(* Logix 5000 project; controller MetsoFilter vendor 1 type 14 code 106 rev 32.11; software revision 32.00 *)

TASK MainTask (continuous, watchdog 500 ms) : MainProgram

MODULES
   Local : vendor 1 type 14 code 106 (Compact 0, rev 32.11)
END_MODULES

TYPE Status_Cycle :   // Status for Each Cycle
STRUCT
   Start_Time : STRING;   // Start Time of Cycle HH:MM
   Cycle_Time : INT;   // Cycle Time in Seconds
   Press_Weight : INT;   // Press wieght of Cycle in Kg
   Pump_Time : INT;   // Pump time in Seconds
   Drying_Time : INT;   // Drying time in Seconds
END_STRUCT
END_TYPE

TYPE Status_Day :   // Status for Each Day
STRUCT
   Date : STRING;   // Days Date
   Total_Tons : REAL;   // Total Tons for the Day
   Shift1_Tons : REAL;   // Shift #1 tons
   Shift2_Tons : REAL;   // Shift #2 Tons
   Shift3_Tons : REAL;   // Shift #3 tons
END_STRUCT
END_TYPE

VAR_GLOBAL   (* controller tags *)
   Alarm_Hatches : BOOL;   // Hatches have taken too long to open or close
   AlarmHornPulser : BOOL;   // Pulse Horn during a new alarm
   AlarmReset : BOOL;   // Alarm Rest Relay
   ALM_AirAndWaterOK_T : TIMER;   // Air and Water OK, Enable Air & Water Valves Alarms
   ALM_DryAir : BOOL;   // Dry Air Not OK
   ALM_LowBattery : BOOL;   // Low Battery Alarm
   ALM_W1 : DINT;   // Alarms to HMI, Word #1
        .1   // Slurry System Not OK
        .0   // Drying Air Not OK
        .2   // Wash Water System Not OK
        .3   // High Pressure Pump Motor Overload
        .4   // Low Pressure Pump Motor Overload
        .5   // Slurry Valve, V1, Failed to Open
        .6   // Slurry Valve, V1, Failed to Close
        .7   // SpareValve, V2, Failed to Open
        .8   // SpareValve, V2, Failed to Close
        .9   // Filtrate Valve, V3, Failed to Open
        .10   // Filtrate Valve, V3, Failed to Close
        .13   // Drying Air Valve, V5, Failed to Open
        .14   // Drying Air Valve, V5, Failed to Close
        .15   // Top Blow AirValve, V6, Failed to Open
        .16   // Top Blow AirValve, V6, Failed to Close
        .17   // Membrane Air Valve, V7, Failed to Open
        .18   // Membrane Air Valve, V7, Failed to Close
        .19   // Top Blow WaterValve, V8, Failed to Open
        .20   // Top Blow Water Valve, V8, Failed to Close
        .21   // Wash WaterValve, V9, Failed to Open
        .22   // Wash WaterValve, V9, Failed to Close
        .23   // Membrane DrainValve, V10, Failed to Open
        .24   // Membrane DrainValve, V10, Failed to Close
        .25   // Upper Hatch Failed to Raise
        .26   // Upper Hatch Failed to Lower
        .27   // Lower Hatch Failed to Raise
        .28   // Lower Hatch Failed to Lower
        .29   // Press Failed to Go to Neutral Position
        .30   // Press Failed to Go to ParkPosition
        .31   // Press Failed to Go to PressPosition
        .11   // Slurry Return Valve, V4, Failed to Open
        .12   // Slurry Return Valve, V4, Failed to Close
   ALM_W2 : DINT;   // Alarms to HMI, Word #2
        .2   // Cloth Dammage
        .0   // Press Weight Sensor Out Of Range
        .1   // Press Pressure Sensor Out Of Range
        .3   // Vibrator Motor Overload
   AlwaysOff : BOOL;   // Always Off Bit
   AS_AirDry : BOOL;   // Auto Sequence, Air Dry
   AS_AirDry_T : TIMER := (PRE := 1000);   // Auto Sequence, Air Dry Timer
   AS_ClothFlush : BOOL;   // Auto Sequence Flush out Cloth
   AS_ClothFlush_T : TIMER := (PRE := 1000);   // Auto Sequence Flush out Cloth Timer
   AS_ClothVibWash : BOOL;   // Auto Sequence Vibrate & Wash Cloth
   AS_ClothVibWash_T : TIMER := (PRE := 1000);   // Auto Sequence Vibrate & Wash Cloth Timer
   AS_Done : BOOL;   // Automatic Sequence Done, Reset Sequence for Next Run
   AS_Drain : BOOL;   // Auto Sequence, Drain
   AS_Drain_T : TIMER := (PRE := 1000);   // Auto Sequence, Drain Timer
   AS_EmptyWeightIsHigh : BOOL;   // Auto Sequence, Empty Wieght is too High
   AS_FeedFilter : BOOL;   // Auto Sequence, Feed Filter
   AS_FeedFilter_T : TIMER := (PRE := 1000);   // Auto Sequence, Feed Filter Timer
   AS_FF_Repeat : BOOL;   // Auto Sequence, Feed Filter has been Repeated at least once
   AS_FF_WeightOK : BOOL;   // Auto Sequence, Feed Filter Weight is OK
   AS_HighEmptyAck : BOOL;   // Auto Sequence High Empty Weight Alarm Acknowlege
   AS_HighEmptyWeight : BOOL;   // Auto Sequence, High Empty Weight, Manually Shake filter
   AS_HighPressClose : BOOL;   // Auto Sequence, Close Press at High Pressure
   AS_HPC_Close_Vx_T : TIMER := (PRE := 1000);   // Auto Sequence, Close ?? Valve Vx Timer
   AS_HPC_Open_V1_T : TIMER := (PRE := 1000);   // Auto Sequence, Open Slurry Valve V1 Timer
   AS_LowFeedAck : BOOL;   // Auto Sequence, Low Feed Weight Alarm Acknowlege
   AS_LowFeedWeight : BOOL;   // Auto Sequence, Low Feed Weight, Enable Retry
   AS_LowPressClose : BOOL;   // Auto Sequence, Close Press at Low Pressure
   AS_LowPressClose_T : TIMER := (PRE := 1000);   // Auto Sequence, Low Pressure Close Timer
   AS_MembComp : BOOL;   // Auto Sequence, Membrane Compress
   AS_MembComp_Ena : BOOL;   // Auto Sequence, Enable Membrane Compress When in Auto Run
   AS_MembComp_T : TIMER := (PRE := 1000);   // Auto Sequence, Membrane Compress Timer
   AS_ResetFF : BOOL;   // Auto Sequence, Reset Feed Filter Logic to Retry
   AS_TopBlow_Wat : BOOL;   // Auto Sequence, Top Blow Water
   AS_TopBlow_Wat_T : TIMER;   // Auto Sequence, Top Blow Water Timer
   AS_TopBlowAir1 : BOOL;   // Auto Sequence, Top Blow Air #1
   AS_TopBlowAir1_T : TIMER := (PRE := 1000);   // Auto Sequence, Top Blow Air #1 Timer
   AS_TopBlowAir2 : BOOL;   // Auto Sequence, Top Blow Air #2
   AS_TopBlowAir2_T : TIMER := (PRE := 1000);   // Auto Sequence, Top Blow Air #2 Timer
   AS_TopBlowWat : BOOL;   // Automatic Sequence, Top Blow & Water
   AS_TopBlowWat_T : TIMER := (PRE := 1000);   // Automatic Sequence, Top Blow & Water Timer
   AS_VibrateCloth : BOOL;   // Auto Sequence Vibrate Cloth
   AS_VibrateCloth_T : TIMER := (PRE := 1000);   // Auto Sequence Vibrate Cloth Timer
   AS_Wait : BOOL;   // Auto Sequence Wait
   AS_Wait_T : TIMER := (PRE := 1000);   // Auto Sequence Wait Timer
   At_Neutral_Pos_T : TIMER := (PRE := 1000);   // Press At Neutral (Open) Position Timer
   At_Parked_Pos_T : TIMER := (PRE := 1000);   // Press At Parked (Closed) Postion Timer
   Auto_ON : BOOL;   // Auto On Mode
   Auto_Reset : BOOL;   // Reset Auto Sequence Logic Abnormally
   Auto_Run : BOOL;   // Run the Next Step of the Auto Sequence
   AutoSeqStarted : BOOL;   // Auto Sequence Started
   Between_Pk_Neu : BOOL;   // Press Between Park and Neutral
   ClothDamaged_T : TIMER := (PRE := 3000);   // Dammaged Cloth Detection Switch On Plus Time
   Colon_STR : STRING := ':'; {constant}   // Constant Colon String = ":"
   Dash_STR : STRING := '-'; {constant}   // Constant Dash String = "-"
   DateTimeArray : DINT[7];
        [0]   // Year
        [1]   // Month(1-12)
        [2]   // Day(1-31)
        [3]   // Hour(0-23)
        [4]   // Minute(0-59)
        [5]   // Second(0-59)
        [6]   // Microsecond (0-999,999)
   Day_STR : STRING;   // Day String(1-31)
   DD_Cycle_1 : Status_Cycle;   // Cycle 1 At Left Side Of Statistics Screen
   DD_Cycle_2 : Status_Cycle;   // Cycle 2
   DD_Cycle_3 : Status_Cycle;   // Cycle 3
   DD_Cycle_4 : Status_Cycle;   // Cycle 4
   DD_Cycle_5 : Status_Cycle;   // Cycle 5
   DD_Cycle_6 : Status_Cycle;   // Cycle 6
   DD_Cycle_7_Now : Status_Cycle;   // Cycle 7, Now being Updated @ Right Side of Statistics Screen
   DD_CyclesLeft : DINT;   // To HMI, Cycles Left Before Servicing
   DD_CycleTime : DINT;   // To HMI, Current Cycle time
   DD_Date_STR : STRING;   // Date String - YYYY-MM-DD
   DD_Day_1 : Status_Day;   // Status Day 1 At Left Side of Statistics Screen
   DD_Day_2 : Status_Day;   // Status Day 2
   DD_Day_3 : Status_Day;   // Status Day 3
   DD_Day_4 : Status_Day;   // Status Day 4
   DD_Day_5 : Status_Day;   // Status Day 5
   DD_Day_6 : Status_Day;   // Status Day 6
   DD_Day_7_Now : Status_Day;   // Status Day 7, Now Being Updated @ Right Side of Statistics Screen
   DD_LastResetDate_STR : DINT;   // On Statistics Screen, Date when last reset performed
   DD_PressPressure : REAL;   // Press Pressure Data Display
   DD_PressWeight : DINT;   // Press Weight from Analog Input Data Display
   DD_Shift3_End : DINT;   // To HMI, Shift 3 End Hour
   DD_Shift3_Start : DINT;   // To HMI, Shift 3 Start Hour
   DD_Time_STR : STRING;   // Time String = HH:MM
   DD_TotalCycles : DINT;   // To HMI, Total Cycles Performed, since last Reset
   DD_TotalTons : DINT;   // To HMI, Total Tons Pressed from Last Reset
   DE_AirDry : DINT;   // Settings Screen, Air Dry Time Data Entry (Seconds)
   DE_ClothVibrate : DINT;   // Settings Screen, Cloth Vibrate Time Data Entry (Seconds)
   DE_ClothVibWash : DINT;   // Settings Screen, Cloth Vibrate and Wash Time Data Entry (Seconds)
   DE_ClothWash : DINT;   // Settings Screen, Cloth Wash Time Data Entry (Seconds)
   DE_ConvIncSpeed : DINT;   // Special Screen, Conv. Inc Speed Data Entry
   DE_DelayedStart : DINT;   // Settings Screen, Delay Start Wait Time Data Entry (Seconds)
   DE_DerivativeFactor : DINT;   // Special Screen, Derivative FactorData Entry
   DE_DerivativeTime : DINT;   // Special Screen, Derivative Time Data Entry
   DE_DiffOilWt_Op_Cl : DINT;   // Special Screen, Differential Oil Weight Open Close Data Entry
   DE_Drain : DINT;   // Settings Screen, Drain Time Data Entry (Seconds)
   DE_FeedFilter : DINT;   // Settings Screen, Feed Filter Time Data Entry (Seconds)
   DE_MembComp : DINT;   // Settings Screen, Membrane Compress Time Data Entry (Seconds)
   DE_MinPressWeight : DINT;   // Special Screen, Minimum Press Weight Data Entry
   DE_MinPresWeight : DINT;   // Special Screen, Minimum Pressure Weight Data Entry
   DE_PressEmptyWeight : DINT;   // Special Screen, Press Empty Weight Data Entry
   DE_ServiceCycles : DINT;   // Special Screen, Service Cycles for Maintenance Data Entry
   DE_Shift1_Start : DINT;   // Special Screen, Shift1 Start Hour, Data Entry
   DE_Shift2_Start : DINT;   // Special Screen, Shift 2 Start Data Entry
   DE_TopBlow2Air1 : DINT;   // Settings Screen, Top Blow Air 1 Time Data Entry (Seconds)
   DE_TopBlow2Air2 : DINT;   // Settings Screen, Top Blow Air 2 Time Data Entry (Seconds)
   DE_TopBlow2Water : DINT;   // Settings Screen, Top Blow Water Time Data Entry (Seconds)
   DryAirSwitch : BOOL;   // Drying Air OK Switch
   DSH1 : BOOL;   // Dammaged Cloth Detection Switch
   DummyInput : BOOL;   // Dummy Input for Temp Inputs File
   DummyInputDINT : DINT;   // Dummy Input from Analog Module
   DummyOutput : BOOL;   // Dummy Output for Temporary outputs File
   Goto_Neutral_T : TIMER := (PRE := 3000);   // Manual / Auto Open (Goto Neutral) Press On Plus Time
   Goto_Park_T : TIMER := (PRE := 3000);   // Go to Park On Plus Time
   Goto_Press_T : TIMER := (PRE := 3000);   // Go to Press Position Output On Plus Time
   GS3 : BOOL;   // Press At Park Position Prox Switch
   GS4 : BOOL;   // Press At Neutral Position Prox Switch
   GS8 : BOOL;   // Press At Press Position Prox Switch
   GSC11 : BOOL;   // Upper Hatch is Closed Proximity Switch
   GSC9 : BOOL;   // Lower Hatch is Closed Proximity Switch
   GSO10 : BOOL;   // Lower Hatch is Open Proximity Switch
   GSO12 : BOOL;   // Upper Hatch is Open Proximity Switch
   H1b : BOOL;   // Hydraulic Valve, Main Drainage
   H2a : BOOL;   // Hydraulic Valve, High Pressure Drainage
   H2b : BOOL;   // Hydraulic Valve, High Pressure Close
   H3a : BOOL;   // Hydraulic Valve, Press Close
   H3b : BOOL;   // Hydraulic Valve, Press Open
   H4a : BOOL;   // Hydraulic Valve, Raise (Open) Lower Hatch
   H4a_On_T : TIMER := (PRE := 3000);   // Hydraulic Valve, Raise (Open) Lower Hatch On Plus Time
   H4b : BOOL;   // Hydraulic Valve, Lower (Close) Lower Hatch
   H4b_On_T : TIMER := (PRE := 3000);   // Hydraulic Valve, Lower (Close) Lower Hatch On Plus Time
   H5a : BOOL;   // Hydraulic Valve, Raise (Open) Upper Hatch
   H5a_On_T : TIMER := (PRE := 3000);   // Hydraulic Valve, Raise (Open) Upper Hatch On Plus Time
   H5b : BOOL;   // Hydraulic Valve, Lower (Close) Upper Hatch
   H5b_On_T : TIMER := (PRE := 3000);   // Hydraulic Valve, Lower (Close) Upper Hatch On Plus Time
   HornPulseDuration_T : TIMER := (PRE := 500);   // Pulse Horn Duration Timer
   HornPulseOff_T : TIMER := (PRE := 500);   // Pulse Horn Off Timer
   HornPulses_C : COUNTER := (PRE := 3);   // Number of times horn pusles for new alarm
   Hour_STR : STRING;   // Hour String(0-23)
   HPP_Run_T : TIMER := (PRE := 3000);   // High Pressure Pump Run Timer
   LPP_Run_T : TIMER := (PRE := 3000);   // Low Pressure Pump Run Timer
   M_HPP_Run : BOOL;   // High Pressure Pump Run Output Bit
   M_HPP_Running : BOOL;   // High Pressure Pump is Running
   M_LPP_Run : BOOL;   // Low Pressure Pump Run Output Bit
   M_LPP_Running : BOOL;   // Low Pressure Pump is Running
   M_Vibrator_Run : BOOL;   // Vibrator Motor Run Output
   M_Vibrator_Run_T : TIMER := (PRE := 3000);   // Vibrator Motor Run Output On Plus Time
   M_Vibrator_Running : BOOL;   // Vibrator Motor Running Input
   MAN_ClosePress : BOOL;   // Manual Close Press to Park Position
   MAN_Vibrate : BOOL;   // Manual Vibrate Flip Flop
   MAN_Wash : BOOL;   // Manual Wash Flip Flop
   Manual_OFF_OSB : BOOL;   // Manual Mode just went Off One Shot
   Manual_ON : BOOL;   // Manual On Mode
   Manual_Operation : BOOL;   // Manual Operation Performed, Reset Auto Sequence
   Manual_OSB : BOOL;   // Manual Pushbutton One shot
   MAS_CloseHatch : BOOL;   // Manual / Auto Close Hatch
   MAS_CloseUpperHatch_T : TIMER := (PRE := 1000);   // Manual / Auto Close Upper Hatch Delay Timer
   MAS_HatchesClosed_T : TIMER := (PRE := 1000);   // Manual / Auto Hatchs are Closed + Time
   MAS_HatchesOpen_T : TIMER := (PRE := 1000);   // Manual / Auto Hatchs are Open + Time
   MAS_OpenHatch : BOOL;   // Manual / Auto Open Hatch
   MAS_OpenLowerHatch_T : TIMER := (PRE := 1000);   // Manual / Auto Open Hatch, Delay Lower Hatch Open
   MAS_OpenPress : BOOL;   // Manual / Auto Open (Goto Neutral) Press
   Minute_STR : STRING;   // Minute String(0-59)
   Month_STR : STRING;   // Month String(1-12)
   MSG_Activity : DINT;   // Activity Message display at left side of the HMI Screens.
   MSG_CloseHatch : BOOL;   // Show Closing Hatches in Sequence & Activity messages latch
   MSG_Main : DINT;   // Main Message at center of screen,
   MSG_MainTemp : DINT;   // Main Message at center of screen, Temporary Holding Register
   MSG_OpenHatch : BOOL;   // Show Opeining Hatch in SEquence & Activity messages latch
   MSG_OpenPress : BOOL;   // Show Opeining Press in Sequence & Activity messages latch
   MSG_SeqTemp : DINT;   // Sequence & Activity Message displays at left side of the HMI Screens, Temp hold
   MSG_Sequence : DINT;   // Sequence Message display at left side of the HMI Screens.
   NewAlarm_OS : BOOL;   // A New Alarm Has Occured
   NewAlarm_PulseHorn : BOOL;   // A New Alarm has Occured, pulse the Horn
   NumberOfAlarms : DINT;   // Number of Active Alarms
   NumberOfAlarms_LS : DINT;   // Number of Active Alarms Last Scan, Detect New Alarm
   OneThirdAir1Preset : DINT;   // 1/3 Top Blow Air 1 time
   OneThirdAir2Preset : DINT;   // 1/3 Top Blow Air 2 time
   PB_AlarmAck : BOOL;   // Alarm Acknowledge Pushbutton
   PB_AlarmReset : BOOL;   // Alarm Reset Pushbutton
   PB_Auto : BOOL;   // Auto Pushbutton
   PB_Auto_Ena : BOOL;   // Auto Pushbutton Enable
   PB_HatchClose : BOOL;   // Hatch Close Pushbutton
   PB_HatchClose_Ena : BOOL;   // Hatch Close Pushbutton Enable
   PB_HatchOpen : BOOL;   // Hatch Open Pushbutton
   PB_HatchOpen_Ena : BOOL;   // Hatch Open Pushbutton Enable
   PB_Manual : BOOL;   // Manual Push Button
   PB_Manual_OS : BOOL;   // Manual Pushbutton One shot
   PB_NextStep : BOOL;   // Next Step Pushbutton
   PB_NextStep_Ena : BOOL;   // Next Step Pushbutton Enable
   PB_PressClose : BOOL;   // Press Close Pushbutton
   PB_PressClose_Ena : BOOL;   // Press Close Pushbutton Enable
   PB_PressOpen : BOOL;   // Press Open Pushbutton
   PB_PressOpen_Ena : BOOL;   // Press Open Pushbutton Enable
   PB_RedoFeed : BOOL;   // Redo Feed Pushbutton
   PB_RedoFeed_Ena : BOOL;   // Redo Feed Pushbutton Enable
   PB_Remote : BOOL;   // Remote Pushbutton Enable
   PB_Remote_Ena : BOOL;   // Remote Pushbutton Enable
   PB_ResetSpecial : BOOL;   // Reset Pushbutton on the Specal Screen, Reset Total Cycles & Weight
   PB_Stop : BOOL;   // Stop Pushbutton
   PB_Stop_Ena : BOOL;   // Stop Pushbutton Enable
   PB_ToNeutral : BOOL;   // To Neutral Pushbutton
   PB_ToNeutral_Ena : BOOL;   // To Neutral Pushbutton Enable
   PB_ToPark : BOOL;   // To Park Pushbutton
   PB_ToPark_Ena : BOOL;   // To Park Pushbutton Enable
   PB_Vibrate : BOOL;   // Vibrate Pushbutton
   PB_Vibrate_Ena : BOOL;   // Vibrate Pushbutton Enable
   PB_Vibrate_OS : BOOL;   // Manual Vibrate Pushbutton One Shot
   PB_Vibrate_OSB : BOOL;   // Manual Vibrate Pushbutton One Shot
   PB_Wash : BOOL;   // Wash Pushbutton
   PB_Wash_Ena : BOOL;   // Wash Pushbutton Enable
   PB_Wash_OS : BOOL;   // Manual Wash Pushbutton One Shot
   PB_Wash_OSB : BOOL;   // Manual Wash Pushbutton One Shot
   Pipe10_Color : DINT;   // Pipe 10 Tag, Slurry Feed, On main Screen
   Pipe1_Color : DINT;   // Pipe 1 at top of main Screen, Main Air Feed
   Pipe2_Color : DINT;   // Pipe 2, below V7, On main Screen
   Pipe3_Color : DINT;   // Pipe 3, below V5, On main Screen
   Pipe4_Color : DINT;   // Pipe 4, Wash, Left of V9, On main Screen
   Pipe5_Color : DINT;   // Pipe 5, Top Blow Water, Left of V8, On main Screen
   Pipe6_Color : DINT;   // Pipe 6, Drain,Below V10, On main Screen
   Pipe7_Color : DINT;   // Pipe 7, Below & Left of V3, On main Screen
   Pipe8_Color : DINT;   // Pipe 8, Connects Slurry Feed and Slurry Return, On main Screen
   Pipe9_Color : DINT;   // Pipe 9 & Tab, Slurry Return, On main Screen
   PLC_Status_Int : INT;   // PLC Status Integer
   PressPressure_OOR_T : TIMER := (PRE := 3000);   // Press Pressure Sensor Out Of Range Plus Time
   PressWeight_OOR_T : TIMER := (PRE := 3000);   // Press Weight Out Of Range Timer
   S_AS_DoneOS : BOOL;   // Statistics, Automatic Sequence Normally Done or Abnormally Stopped One Shot
   S_AS_DoneOSB : BOOL;   // Statistics, Automatic Sequence Done One Shot
   S_AS_StartOS : BOOL;   // Statistics, Automatic Sequence Started One Shot
   S_AS_StartOSB : BOOL;   // Statistics, Automatic Sequence Started One Shot
   S_CloseHatchOSB : BOOL;   // Statistics, Hatch Starting to Close, One Shot
   S_CycleTimer : TIMER := (PRE := 999999999);   // Statistics, Cycle Time Timer
   S_DryingTimer : TIMER := (PRE := 999999999);   // Statistics, Drying Time Timer
   S_LastCycleStopped : BOOL;   // Last Auto Sequence Stopped Abnormally, do not shift Cycles, but cearl cycle 7
   S_NewDay : BOOL;   // Statistics, Midnight & No Sequence Running, Update Days
   S_OpenHatchOSB : BOOL;   // Statistics, Hatch Starting to Open, One Shot
   S_PressWeightTons : REAL;   // Statistics, Weight in Tons Just Pressed
   S_PumpTimer : TIMER := (PRE := 999999999);   // Statistics, Pump Time Timer
   S_Shift1 : BOOL;   // Statistics, Shift 1 in Progress
   S_Shift1_OSB : BOOL;   // Statistics, Start of Shift 1 One shot
   S_Shift2 : BOOL;   // Statistics, Shift 2 in Progress
   S_Shift2_OSB : BOOL;   // Statistics, Start of Shift 2 One shot
   S_Shift3 : BOOL;   // Statistics, Shift 3 in Progress
   S_Shift3_OSB : BOOL;   // Statistics, Start of Shift 3 One shot
   S_TempDINT : DINT;   // Statistics, Tempory Holding DINT
   S_WeightHatchOpen : DINT;   // Statistics, Weight of Press just as hatches Open
   S_ZeroHour_Latch : BOOL;   // Zero Hour Latch, wait for current sequence to finish, if running
   S_ZeroHour_OSB : BOOL;   // Hour = Zero, New Day One Shot
   SlurrySystemSwitch : BOOL;   // Slurry System OK Switch
   TwoThirdsAir1Preset : DINT;   // 2/3 Top Blow Air 1 time
   TwoThirdsAir2Preset : DINT;   // 2/3 Top Blow Air 2 time
   V10_GSC : BOOL;   // Valve #10, Membrane Drain, Closed Input
   V10_GSO : BOOL;   // Valve #10, Membrane Drain, Opened Input
   V10_Off_T : TIMER := (PRE := 3000);   // Valve #10, Membrane Drain, Ouput Bit Off Plus Time, Valve shoud be Open
   V10_On_T : TIMER := (PRE := 3000);   // Valve #10, Membrane Drain, Ouput Bit On Plus Time, Valve shoud be Closed
   V1_GSC : BOOL;   // Valve #1, Slurry Supply, Closed Input
   V1_GSO : BOOL;   // Valve #1, Slurry Supply, Open Input
   V1_Off_T : TIMER := (PRE := 3000);   // Valve #1, Slurry Supply, Open Output Bit Off Plus Time
   V1_On_T : TIMER := (PRE := 3000);   // Valve #1, Slurry Supply, Open Output Bit On Plus Time
   V3_GSC : BOOL;   // Valve #3, Filtrate, Closed Input
   V3_GSO : BOOL;   // Valve #3, Filtrate, Open Input
   V3_Off_T : TIMER := (PRE := 3000);   // Valve #3, Filtrate, Open Output Bit Off Plus time
   V3_On_T : TIMER := (PRE := 3000);   // Valve #3, Filtrate, Open Output Bit On Plus time
   V4_GSC : BOOL;   // Valve #4, Slurry Return, Closed Input
   V4_GSO : BOOL;   // Valve #4, Slurry Return, Open Input
   V4_Off_T : TIMER := (PRE := 3000);   // Valve #4, Slurry Return, Open Output Bit Off Plus Time
   V4_On_T : TIMER := (PRE := 3000);   // Valve #4, Slurry Return, Open Output Bit On Plus Time
   V5_GSC : BOOL;   // Valve #5, Drying Air, Closed Input
   V5_GSO : BOOL;   // Valve #5, Drying Air, Opened Input
   V5_Off_T : TIMER := (PRE := 3000);   // Valve #5, Drying Air, Open Output Bit Off Plus Time
   V5_On_T : TIMER := (PRE := 3000);   // Valve #5, Drying Air, Open Output Bit On Plus Time
   V6_GSC : BOOL;   // Valve #6, Top Blow Air, Closed Input
   V6_GSO : BOOL;   // Valve #6, Top Blow Air, Opened Input
   V6_Off_T : TIMER := (PRE := 3000);   // Valve #6, Top Blow Air, Open Output Bit On Plus Time
   V6_On_T : TIMER := (PRE := 3000);   // Valve #6, Top Blow Air, Open Output Bit On Plus Time
   V7_GSC : BOOL;   // Valve #7, Membrane Air, Closed Input
   V7_GSO : BOOL;   // Valve #7, Membrane Air, Opened Input
   V7_Off_T : TIMER := (PRE := 3000);   // Valve #7, Membrane Air, Open Output Bit Off Plus Time
   V7_On_T : TIMER := (PRE := 3000);   // Valve #7, Membrane Air, Open Output Bit On Plus time
   V8_GSC : BOOL;   // Valve #8, Top Blow Water, Closed Input
   V8_GSO : BOOL;   // Valve #8, Top Blow Water, Opened Input
   V8_Off_T : TIMER := (PRE := 3000);   // Valve #8, Top Blow Water, Open Output Bit Off Plus Time
   V8_On_T : TIMER := (PRE := 3000);   // Valve #8, Top Blow Water, Open Output Bit On Plus Time
   V9_GSC : BOOL;   // Valve #9, Wash Water, Closed Input
   V9_GSO : BOOL;   // Valve #9, Wash Water, Opened Input
   V9_Off_T : TIMER := (PRE := 3000);   // Valve #9, Wash Water, Open Ouput Bit Off Plus Time
   V9_On_T : TIMER := (PRE := 3000);   // Valve #9, Wash Water, Open Ouput Bit On Plus Time
   WashWaterSwitch : BOOL;   // Wash Water System OK Switch
   WaterInfeedColor : DINT;   // Water Infeed Color
   Year_STR : STRING;   // Year String
   YV1 : BOOL;   // Valve #1, Slurry Supply, Open Output Bit
   YV10 : BOOL;   // Valve #10, Membrane Drain, Normally Open, Energize to Close, Output Bit
   YV3 : BOOL;   // Valve #3, Filtrate, Open Output Bit
   YV4 : BOOL;   // Valve #4, Slurry Return, Open Output Bit
   YV5 : BOOL;   // Valve #5, Drying Air, Open Output Bit
   YV6 : BOOL;   // Valve #6, Top Blow Air, Open Output Bit
   YV7 : BOOL;   // Valve #7, Membrane Air, Open Output Bit
   YV8 : BOOL;   // Valve #8, Top Blow Water, Open Output Bit
   YV9 : BOOL;   // Valve #9, Wash Water, Open Ouput Bit
   Zero_STR : STRING := '0'; {constant}   // Constant String= "0" Pad Values <10 0-9 -> 00-09
END_VAR

PROGRAM MainProgram   (* main routine MainRoutine *)

ROUTINE _01_MapInputs   (* ladder *)
// Map PLC Inputs to Input Bits
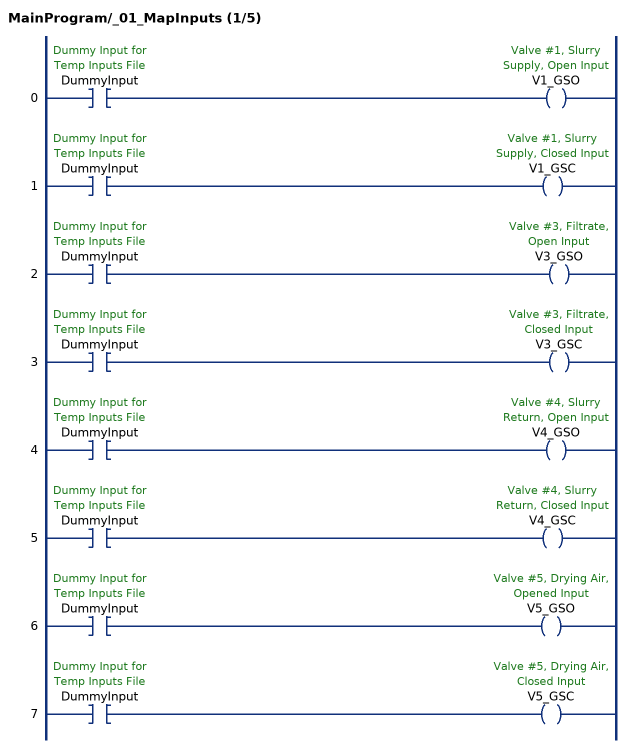
   0: XIC(DummyInput)OTE(V1_GSO);
   1: XIC(DummyInput)OTE(V1_GSC);
   2: XIC(DummyInput)OTE(V3_GSO);
   3: XIC(DummyInput)OTE(V3_GSC);
   4: XIC(DummyInput)OTE(V4_GSO);
   5: XIC(DummyInput)OTE(V4_GSC);
   6: XIC(DummyInput)OTE(V5_GSO);
   7: XIC(DummyInput)OTE(V5_GSC);
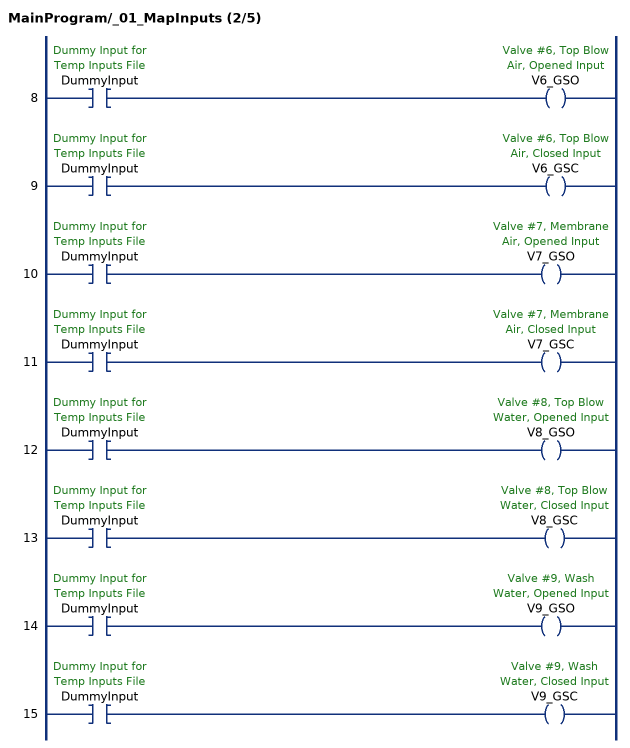
   8: XIC(DummyInput)OTE(V6_GSO);
   9: XIC(DummyInput)OTE(V6_GSC);
   10: XIC(DummyInput)OTE(V7_GSO);
   11: XIC(DummyInput)OTE(V7_GSC);
   12: XIC(DummyInput)OTE(V8_GSO);
   13: XIC(DummyInput)OTE(V8_GSC);
   14: XIC(DummyInput)OTE(V9_GSO);
   15: XIC(DummyInput)OTE(V9_GSC);
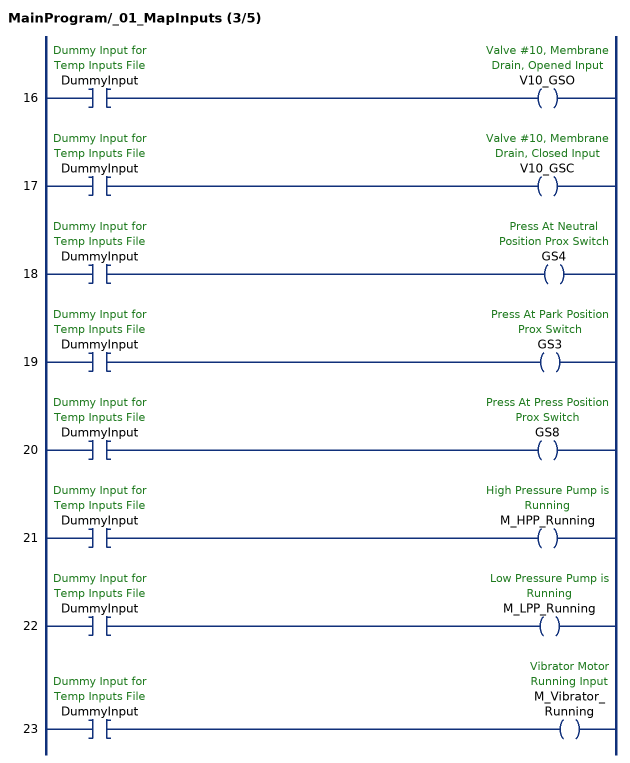
   16: XIC(DummyInput)OTE(V10_GSO);
   17: XIC(DummyInput)OTE(V10_GSC);
   18: XIC(DummyInput)OTE(GS4);
   19: XIC(DummyInput)OTE(GS3);
   20: XIC(DummyInput)OTE(GS8);
   21: XIC(DummyInput)OTE(M_HPP_Running);
   22: XIC(DummyInput)OTE(M_LPP_Running);
   23: XIC(DummyInput)OTE(M_Vibrator_Running);
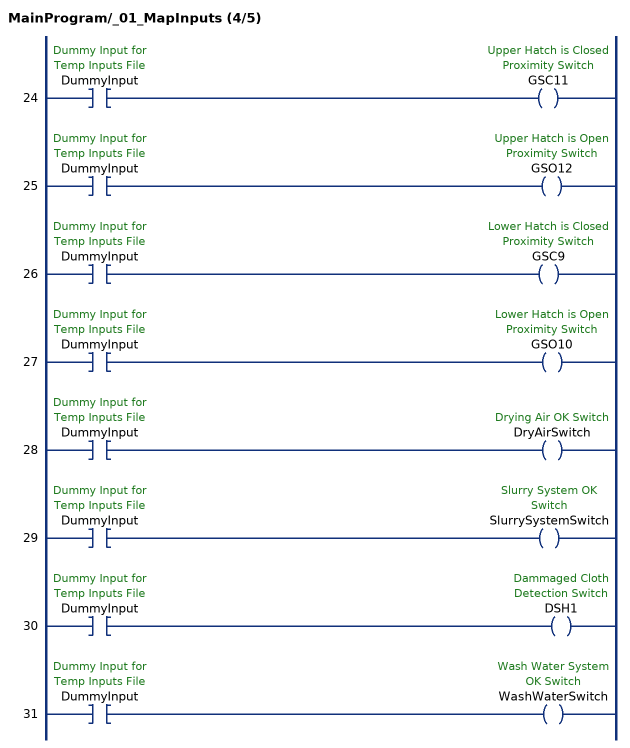
   24: XIC(DummyInput)OTE(GSC11);
   25: XIC(DummyInput)OTE(GSO12);
   26: XIC(DummyInput)OTE(GSC9);
   27: XIC(DummyInput)OTE(GSO10);
   28: XIC(DummyInput)OTE(DryAirSwitch);
   29: XIC(DummyInput)OTE(SlurrySystemSwitch);
   30: XIC(DummyInput)OTE(DSH1);
   31: XIC(DummyInput)OTE(WashWaterSwitch);
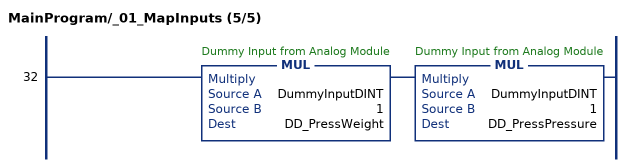
   32: MUL(DummyInputDINT,1,DD_PressWeight)MUL(DummyInputDINT,1,DD_PressPressure);
END_ROUTINE

ROUTINE _02_System_State_Buttons   (* ladder *)
// System State and HMI Button Enables
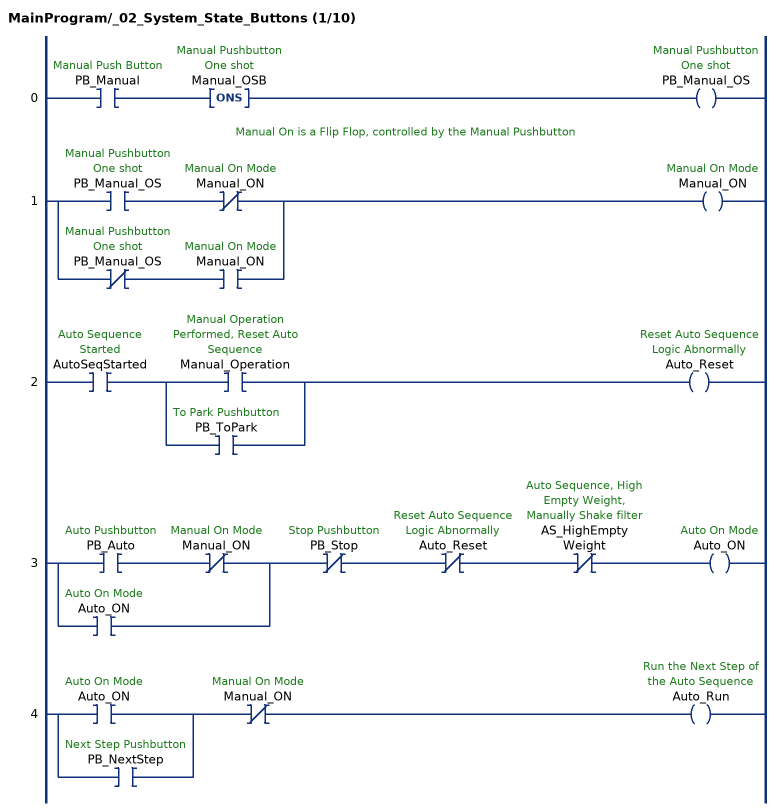
   0: XIC(PB_Manual)ONS(Manual_OSB)OTE(PB_Manual_OS);
   // Manual On is a Flip Flop, controlled by the Manual Pushbutton
   1: [XIC(PB_Manual_OS) XIO(Manual_ON) ,XIO(PB_Manual_OS) XIC(Manual_ON) ]OTE(Manual_ON);
   2: XIC(AutoSeqStarted)[XIC(Manual_Operation) ,XIC(PB_ToPark) ]OTE(Auto_Reset);
   3: [XIC(PB_Auto) XIO(Manual_ON) ,XIC(Auto_ON) ]XIO(PB_Stop)XIO(Auto_Reset)XIO(AS_HighEmptyWeight)OTE(Auto_ON);
   4: [XIC(Auto_ON) ,XIC(PB_NextStep) ]XIO(Manual_ON)OTE(Auto_Run);
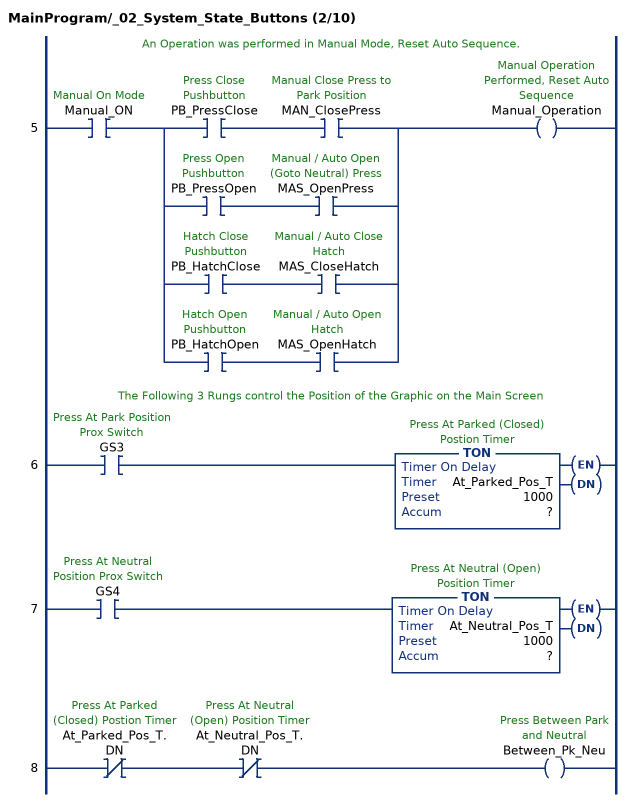
   // An Operation was performed in Manual Mode, Reset Auto Sequence.
   5: XIC(Manual_ON)[XIC(PB_PressClose) XIC(MAN_ClosePress) ,XIC(PB_PressOpen) XIC(MAS_OpenPress) ,XIC(PB_HatchClose) XIC(MAS_CloseHatch) ,XIC(PB_HatchOpen) XIC(MAS_OpenHatch) ]OTE(Manual_Operation);
   // The Following 3 Rungs control the Position of the Graphic on the Main Screen
   6: XIC(GS3)TON(At_Parked_Pos_T,?,?);
   7: XIC(GS4)TON(At_Neutral_Pos_T,?,?);
   8: XIO(At_Parked_Pos_T.DN)XIO(At_Neutral_Pos_T.DN)OTE(Between_Pk_Neu);
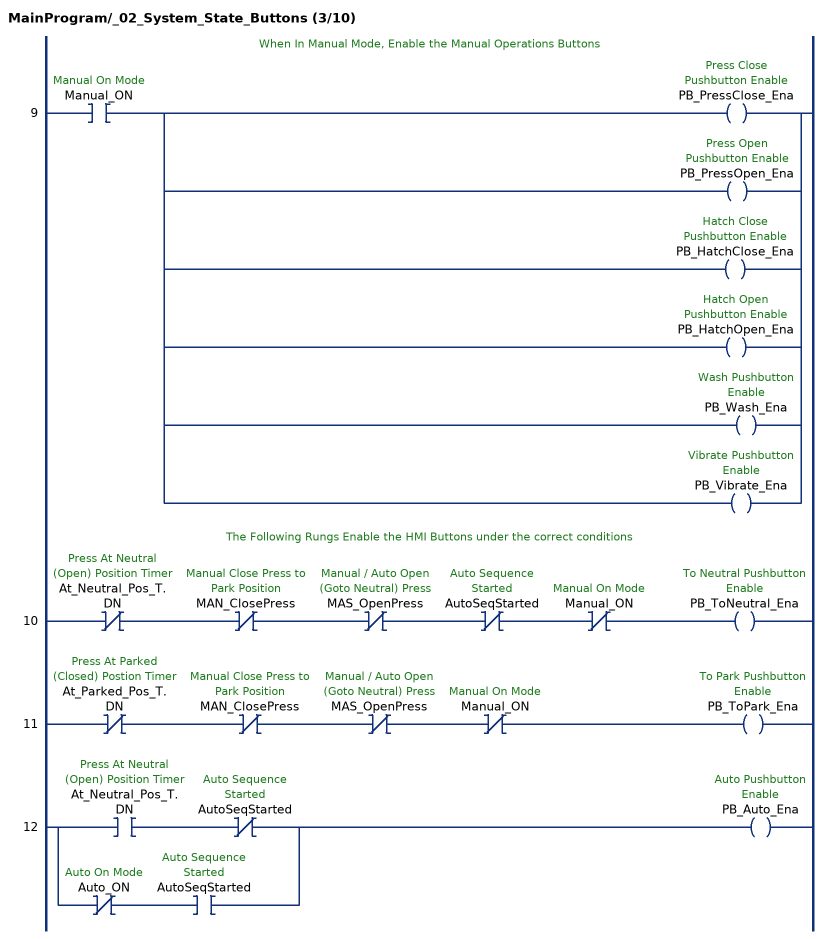
   // When In Manual Mode, Enable the Manual Operations Buttons
   9: XIC(Manual_ON)[OTE(PB_PressClose_Ena) ,OTE(PB_PressOpen_Ena) ,OTE(PB_HatchClose_Ena) ,OTE(PB_HatchOpen_Ena) ,OTE(PB_Wash_Ena) ,OTE(PB_Vibrate_Ena) ];
   // The Following Rungs Enable the HMI Buttons under the correct conditions
   10: XIO(At_Neutral_Pos_T.DN)XIO(MAN_ClosePress)XIO(MAS_OpenPress)XIO(AutoSeqStarted)XIO(Manual_ON)OTE(PB_ToNeutral_Ena);
   11: XIO(At_Parked_Pos_T.DN)XIO(MAN_ClosePress)XIO(MAS_OpenPress)XIO(Manual_ON)OTE(PB_ToPark_Ena);
   12: [XIC(At_Neutral_Pos_T.DN) XIO(AutoSeqStarted) ,XIO(Auto_ON) XIC(AutoSeqStarted) ]OTE(PB_Auto_Ena);
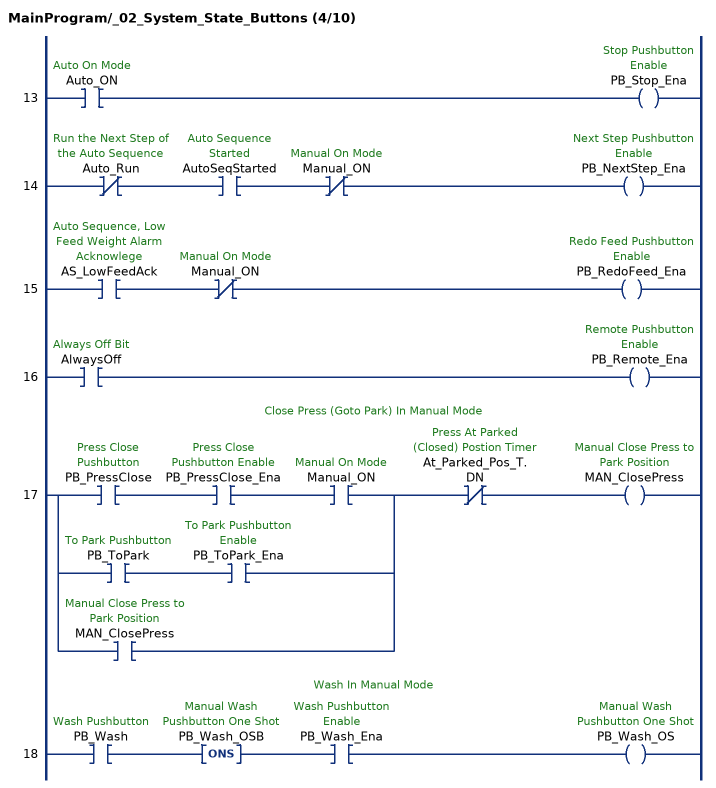
   13: XIC(Auto_ON)OTE(PB_Stop_Ena);
   14: XIO(Auto_Run)XIC(AutoSeqStarted)XIO(Manual_ON)OTE(PB_NextStep_Ena);
   15: XIC(AS_LowFeedAck)XIO(Manual_ON)OTE(PB_RedoFeed_Ena);
   16: XIC(AlwaysOff)OTE(PB_Remote_Ena);
   // Close Press (Goto Park) In Manual Mode
   17: [XIC(PB_PressClose) XIC(PB_PressClose_Ena) XIC(Manual_ON) ,XIC(PB_ToPark) XIC(PB_ToPark_Ena) ,XIC(MAN_ClosePress) ]XIO(At_Parked_Pos_T.DN)OTE(MAN_ClosePress);
   // Wash In Manual Mode
   18: XIC(PB_Wash)ONS(PB_Wash_OSB)XIC(PB_Wash_Ena)OTE(PB_Wash_OS);
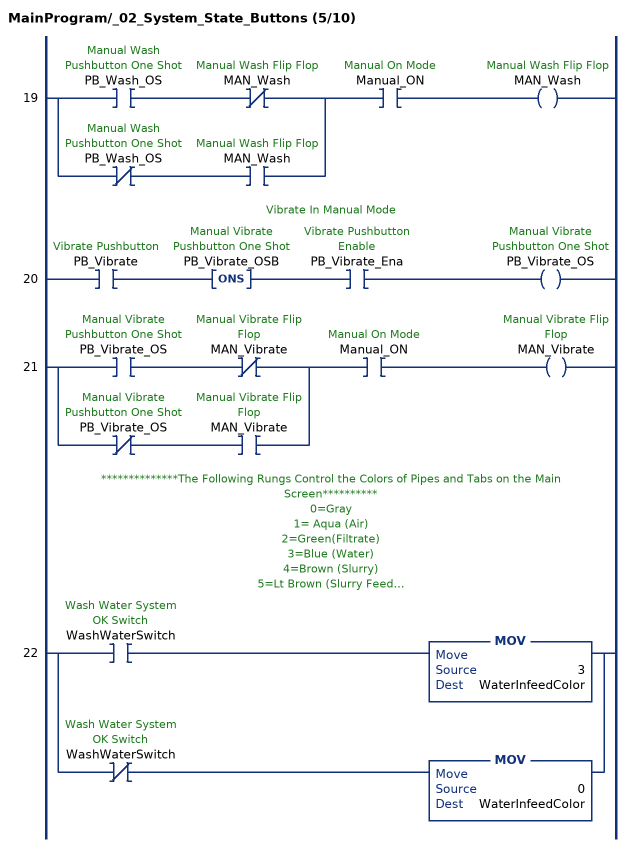
   19: [XIC(PB_Wash_OS) XIO(MAN_Wash) ,XIO(PB_Wash_OS) XIC(MAN_Wash) ]XIC(Manual_ON)OTE(MAN_Wash);
   // Vibrate In Manual Mode
   20: XIC(PB_Vibrate)ONS(PB_Vibrate_OSB)XIC(PB_Vibrate_Ena)OTE(PB_Vibrate_OS);
   21: [XIC(PB_Vibrate_OS) XIO(MAN_Vibrate) ,XIO(PB_Vibrate_OS) XIC(MAN_Vibrate) ]XIC(Manual_ON)OTE(MAN_Vibrate);
   // **************The Following Rungs Control the Colors of Pipes and Tabs on the Main Screen**********
   // 0=Gray
   // 1= Aqua (Air)
   // 2=Green(Filtrate)
   // 3=Blue (Water)
   // 4=Brown (Slurry)
   // 5=Lt Brown (Slurry Feed)
   // Water Infeed Short Pipes & Tabs
   22: [XIC(WashWaterSwitch) MOV(3,WaterInfeedColor) ,XIO(WashWaterSwitch) MOV(0,WaterInfeedColor) ];
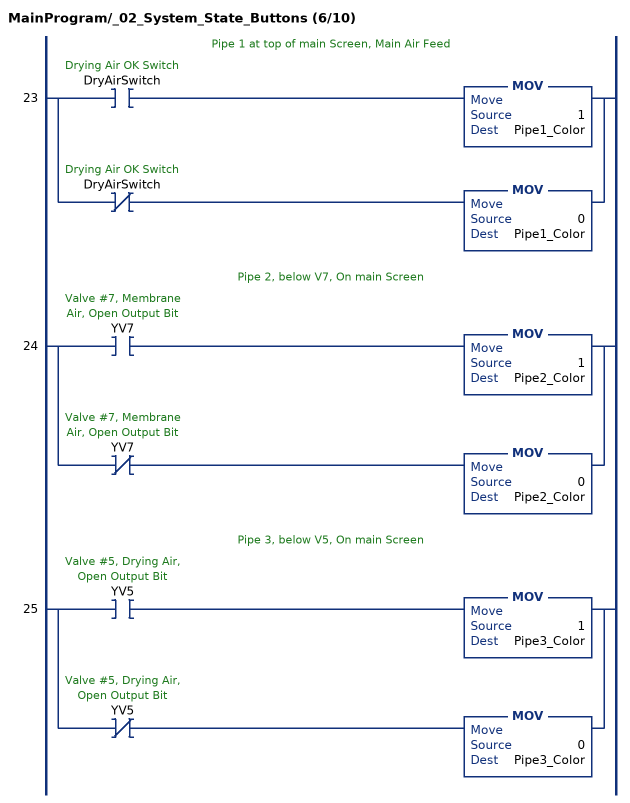
   // Pipe 1 at top of main Screen, Main Air Feed
   23: [XIC(DryAirSwitch) MOV(1,Pipe1_Color) ,XIO(DryAirSwitch) MOV(0,Pipe1_Color) ];
   // Pipe 2, below V7, On main Screen
   24: [XIC(YV7) MOV(1,Pipe2_Color) ,XIO(YV7) MOV(0,Pipe2_Color) ];
   // Pipe 3, below V5, On main Screen
   25: [XIC(YV5) MOV(1,Pipe3_Color) ,XIO(YV5) MOV(0,Pipe3_Color) ];
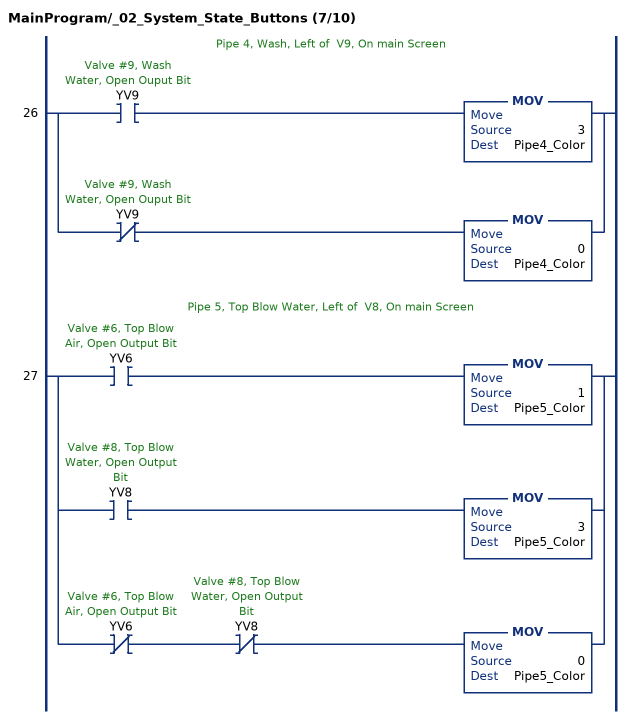
   // Pipe 4, Wash, Left of  V9, On main Screen
   26: [XIC(YV9) MOV(3,Pipe4_Color) ,XIO(YV9) MOV(0,Pipe4_Color) ];
   // Pipe 5, Top Blow Water, Left of  V8, On main Screen
   27: [XIC(YV6) MOV(1,Pipe5_Color) ,XIC(YV8) MOV(3,Pipe5_Color) ,XIO(YV6) XIO(YV8) MOV(0,Pipe5_Color) ];
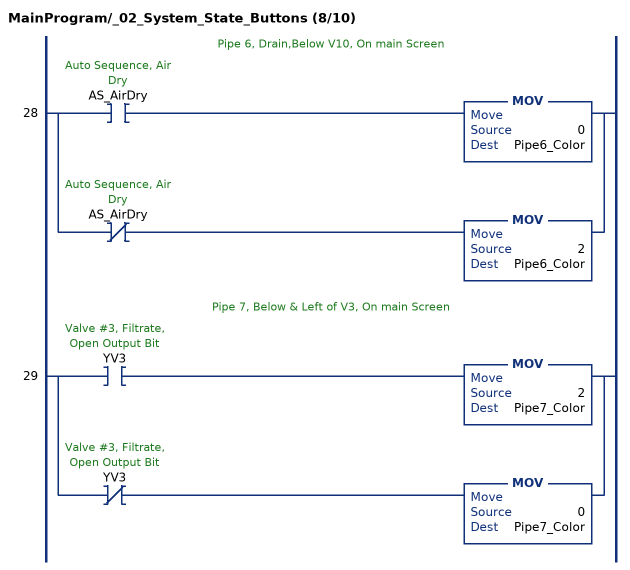
   // Pipe 6, Drain,Below V10, On main Screen
   28: [XIC(AS_AirDry) MOV(0,Pipe6_Color) ,XIO(AS_AirDry) MOV(2,Pipe6_Color) ];
   // Pipe 7, Below & Left of V3, On main Screen
   29: [XIC(YV3) MOV(2,Pipe7_Color) ,XIO(YV3) MOV(0,Pipe7_Color) ];
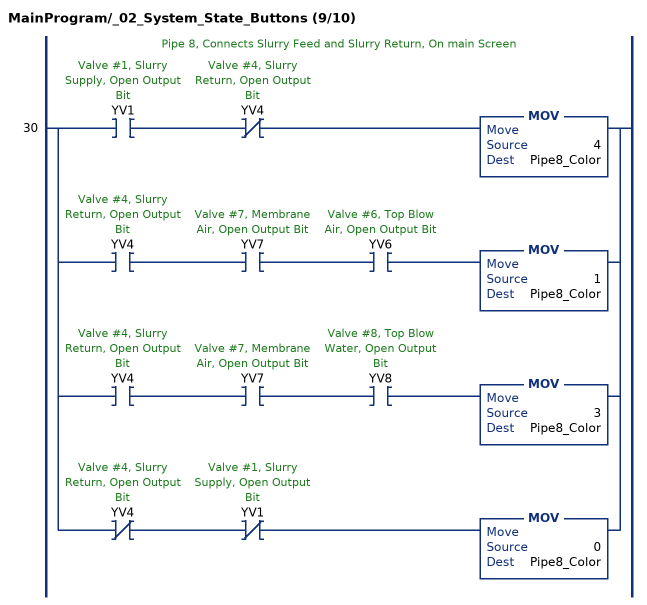
   // Pipe 8, Connects Slurry Feed and Slurry Return, On main Screen
   30: [XIC(YV1) XIO(YV4) MOV(4,Pipe8_Color) ,XIC(YV4) XIC(YV7) XIC(YV6) MOV(1,Pipe8_Color) ,XIC(YV4) XIC(YV7) XIC(YV8) MOV(3,Pipe8_Color) ,XIO(YV4) XIO(YV1) MOV(0,Pipe8_Color) ];
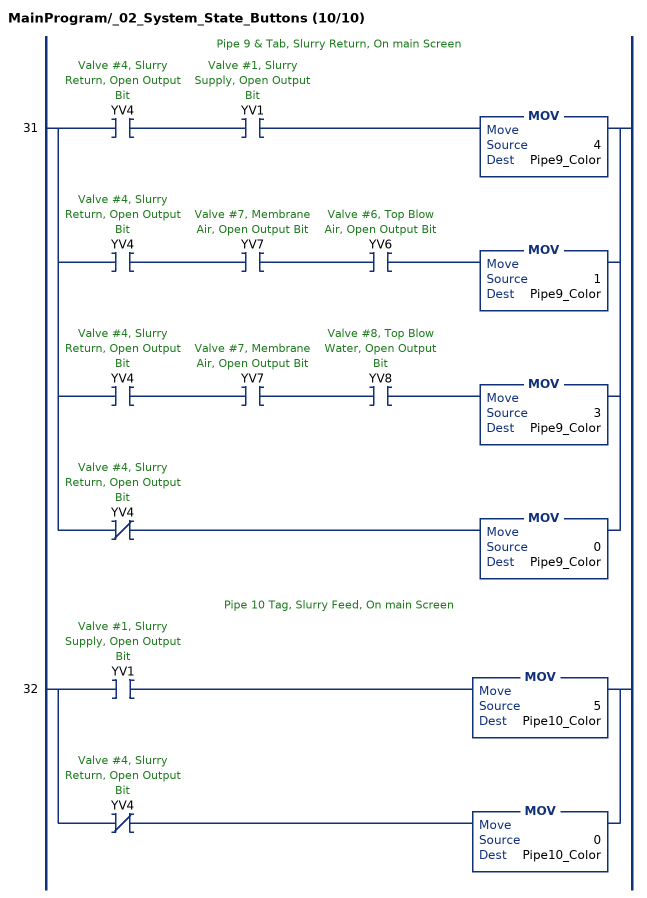
   // Pipe 9 & Tab, Slurry Return, On main Screen
   31: [XIC(YV4) XIC(YV1) MOV(4,Pipe9_Color) ,XIC(YV4) XIC(YV7) XIC(YV6) MOV(1,Pipe9_Color) ,XIC(YV4) XIC(YV7) XIC(YV8) MOV(3,Pipe9_Color) ,XIO(YV4) MOV(0,Pipe9_Color) ];
   // Pipe 10 Tag, Slurry Feed, On main Screen
   32: [XIC(YV1) MOV(5,Pipe10_Color) ,XIO(YV4) MOV(0,Pipe10_Color) ];
END_ROUTINE

ROUTINE _03_Automatic_Sequence   (* ladder *)
// Automatic Sequence Relays
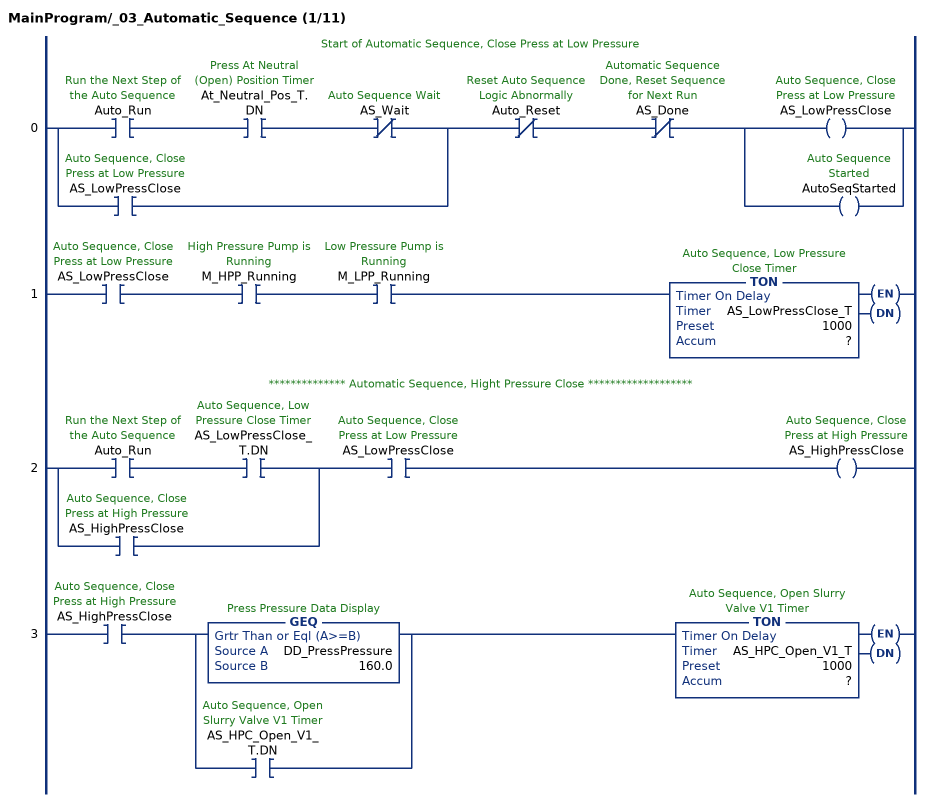
   // Start of Automatic Sequence, Close Press at Low Pressure
   0: [XIC(Auto_Run) XIC(At_Neutral_Pos_T.DN) XIO(AS_Wait) ,XIC(AS_LowPressClose) ]XIO(Auto_Reset)XIO(AS_Done)[OTE(AS_LowPressClose) ,OTE(AutoSeqStarted) ];
   1: XIC(AS_LowPressClose)XIC(M_HPP_Running)XIC(M_LPP_Running)TON(AS_LowPressClose_T,?,?);
   // ************** Automatic Sequence, Hight Pressure Close *******************
   2: [XIC(Auto_Run) XIC(AS_LowPressClose_T.DN) ,XIC(AS_HighPressClose) ]XIC(AS_LowPressClose)OTE(AS_HighPressClose);
   3: XIC(AS_HighPressClose)[GEQ(DD_PressPressure,160.0) ,XIC(AS_HPC_Open_V1_T.DN) ]TON(AS_HPC_Open_V1_T,?,?);
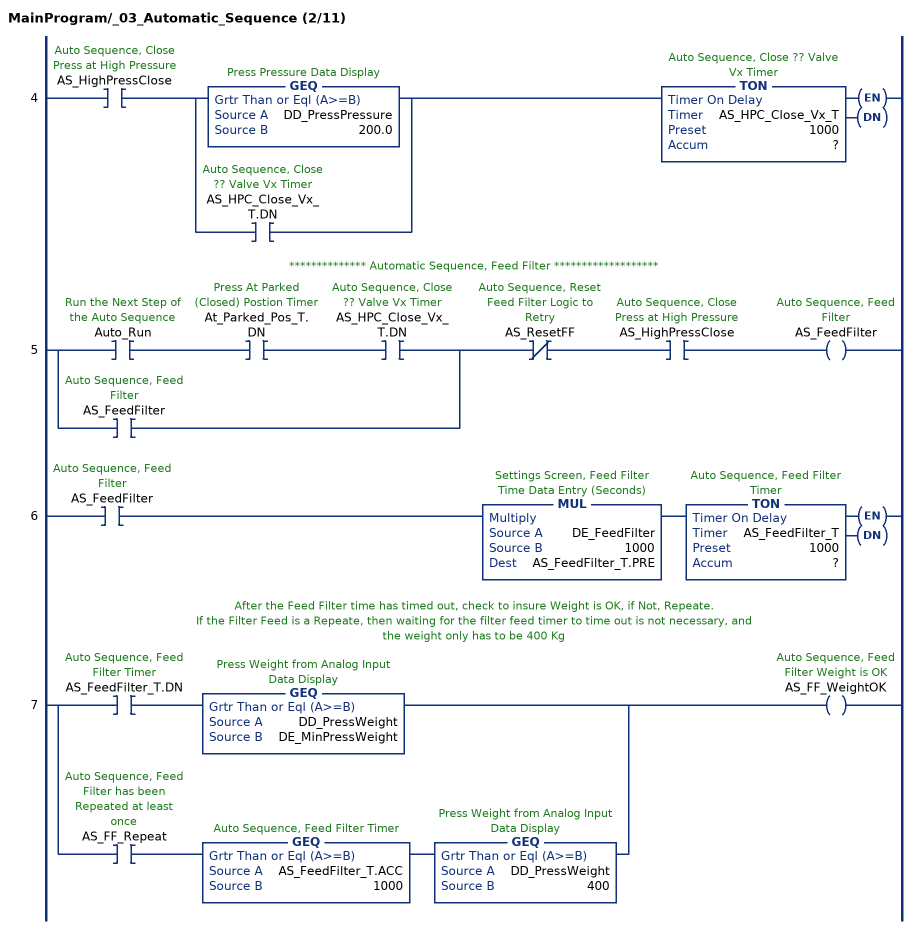
   4: XIC(AS_HighPressClose)[GEQ(DD_PressPressure,200.0) ,XIC(AS_HPC_Close_Vx_T.DN) ]TON(AS_HPC_Close_Vx_T,?,?);
   // ************** Automatic Sequence, Feed Filter *******************
   5: [XIC(Auto_Run) XIC(At_Parked_Pos_T.DN) XIC(AS_HPC_Close_Vx_T.DN) ,XIC(AS_FeedFilter) ]XIO(AS_ResetFF)XIC(AS_HighPressClose)OTE(AS_FeedFilter);
   6: XIC(AS_FeedFilter)MUL(DE_FeedFilter,1000,AS_FeedFilter_T.PRE)TON(AS_FeedFilter_T,?,?);
   // After the Feed Filter time has timed out, check to insure Weight is OK, if Not, Repeate.
   // If the Filter Feed is a Repeate, then waiting for the filter feed timer to time out is not necessary, and
   // the weight only has to be 400 Kg
   7: [XIC(AS_FeedFilter_T.DN) GEQ(DD_PressWeight,DE_MinPressWeight) ,XIC(AS_FF_Repeat) GEQ(AS_FeedFilter_T.ACC,1000) GEQ(DD_PressWeight,400) ]OTE(AS_FF_WeightOK);
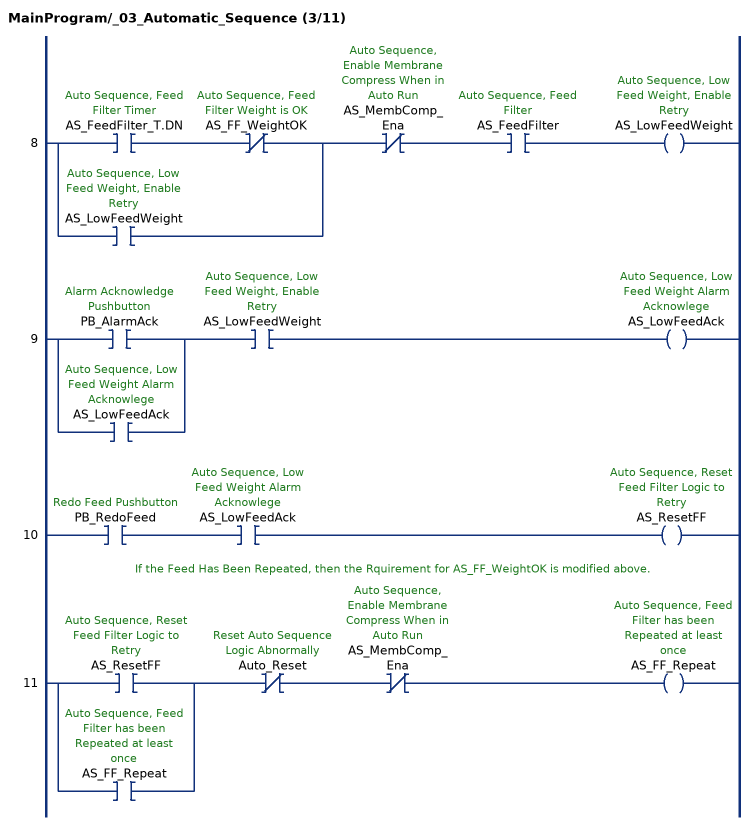
   8: [XIC(AS_FeedFilter_T.DN) XIO(AS_FF_WeightOK) ,XIC(AS_LowFeedWeight) ]XIO(AS_MembComp_Ena)XIC(AS_FeedFilter)OTE(AS_LowFeedWeight);
   9: [XIC(PB_AlarmAck) ,XIC(AS_LowFeedAck) ]XIC(AS_LowFeedWeight)OTE(AS_LowFeedAck);
   10: XIC(PB_RedoFeed)XIC(AS_LowFeedAck)OTE(AS_ResetFF);
   // If the Feed Has Been Repeated, then the Rquirement for AS_FF_WeightOK is modified above.
   11: [XIC(AS_ResetFF) ,XIC(AS_FF_Repeat) ]XIO(Auto_Reset)XIO(AS_MembComp_Ena)OTE(AS_FF_Repeat);
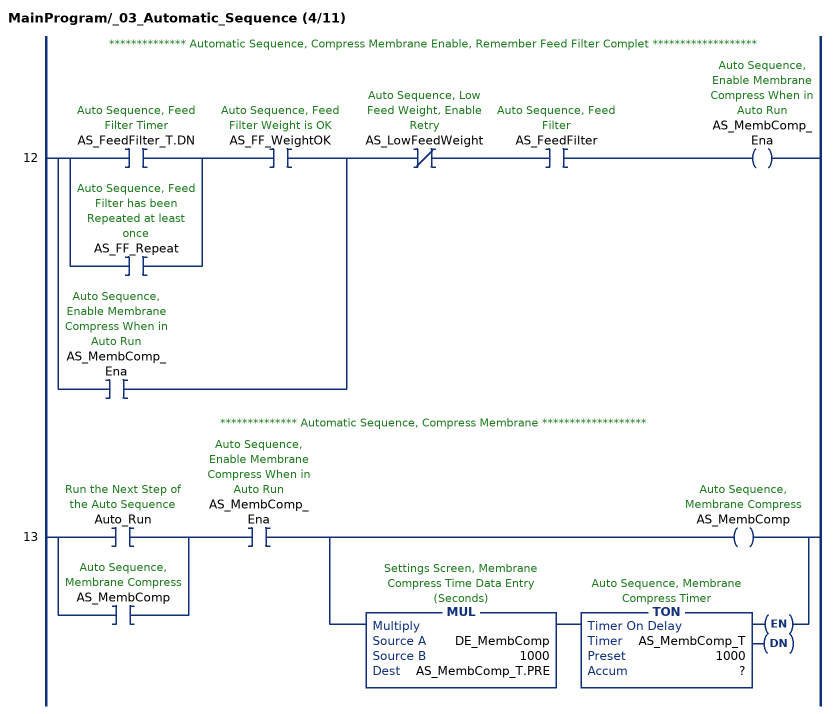
   // ************** Automatic Sequence, Compress Membrane Enable, Remember Feed Filter Complet *******************
   12: [[XIC(AS_FeedFilter_T.DN) ,XIC(AS_FF_Repeat) ] XIC(AS_FF_WeightOK) ,XIC(AS_MembComp_Ena) ]XIO(AS_LowFeedWeight)XIC(AS_FeedFilter)OTE(AS_MembComp_Ena);
   // ************** Automatic Sequence, Compress Membrane *******************
   13: [XIC(Auto_Run) ,XIC(AS_MembComp) ]XIC(AS_MembComp_Ena)[OTE(AS_MembComp) ,MUL(DE_MembComp,1000,AS_MembComp_T.PRE) TON(AS_MembComp_T,?,?) ];
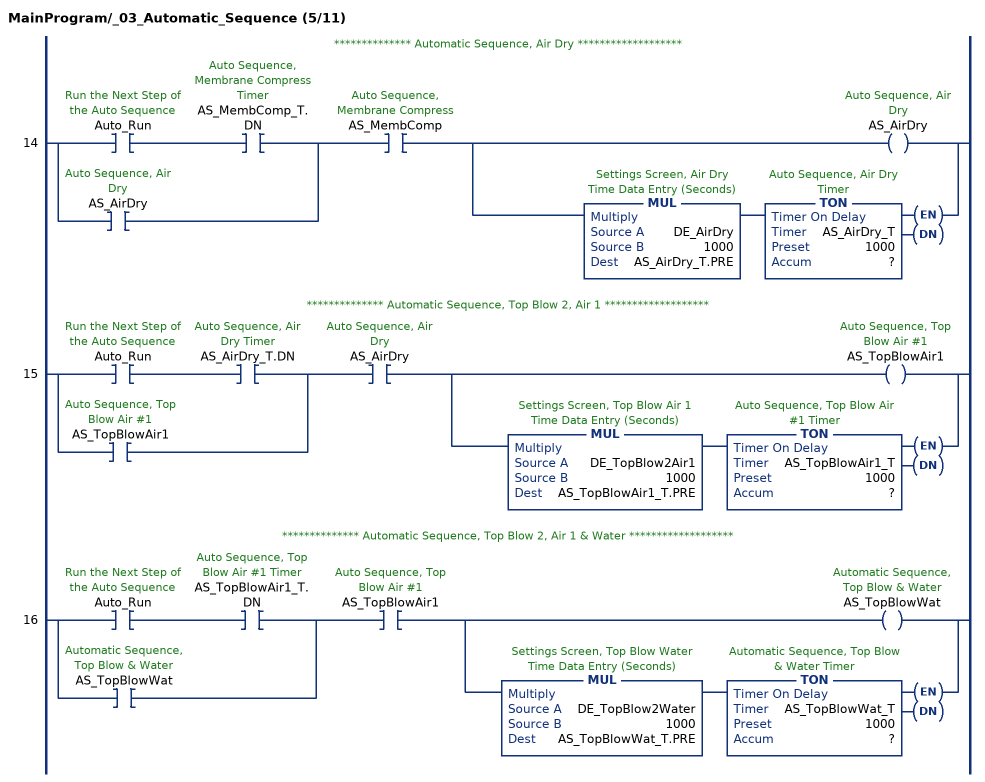
   // ************** Automatic Sequence, Air Dry *******************
   14: [XIC(Auto_Run) XIC(AS_MembComp_T.DN) ,XIC(AS_AirDry) ]XIC(AS_MembComp)[OTE(AS_AirDry) ,MUL(DE_AirDry,1000,AS_AirDry_T.PRE) TON(AS_AirDry_T,?,?) ];
   // ************** Automatic Sequence, Top Blow 2, Air 1 *******************
   15: [XIC(Auto_Run) XIC(AS_AirDry_T.DN) ,XIC(AS_TopBlowAir1) ]XIC(AS_AirDry)[OTE(AS_TopBlowAir1) ,MUL(DE_TopBlow2Air1,1000,AS_TopBlowAir1_T.PRE) TON(AS_TopBlowAir1_T,?,?) ];
   // ************** Automatic Sequence, Top Blow 2, Air 1 & Water *******************
   16: [XIC(Auto_Run) XIC(AS_TopBlowAir1_T.DN) ,XIC(AS_TopBlowWat) ]XIC(AS_TopBlowAir1)[OTE(AS_TopBlowWat) ,MUL(DE_TopBlow2Water,1000,AS_TopBlowWat_T.PRE) TON(AS_TopBlowWat_T,?,?) ];
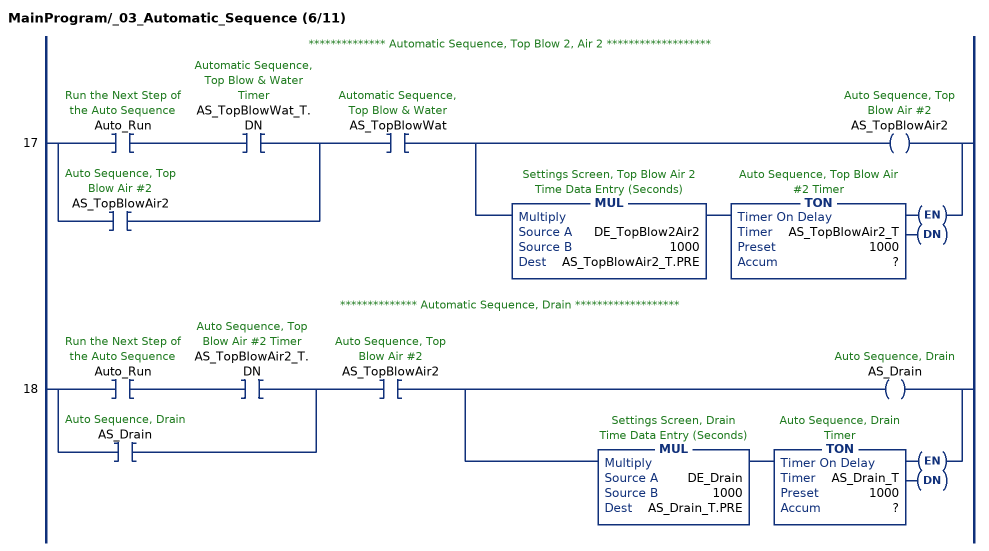
   // ************** Automatic Sequence, Top Blow 2, Air 2 *******************
   17: [XIC(Auto_Run) XIC(AS_TopBlowWat_T.DN) ,XIC(AS_TopBlowAir2) ]XIC(AS_TopBlowWat)[OTE(AS_TopBlowAir2) ,MUL(DE_TopBlow2Air2,1000,AS_TopBlowAir2_T.PRE) TON(AS_TopBlowAir2_T,?,?) ];
   // ************** Automatic Sequence, Drain *******************
   18: [XIC(Auto_Run) XIC(AS_TopBlowAir2_T.DN) ,XIC(AS_Drain) ]XIC(AS_TopBlowAir2)[OTE(AS_Drain) ,MUL(DE_Drain,1000,AS_Drain_T.PRE) TON(AS_Drain_T,?,?) ];
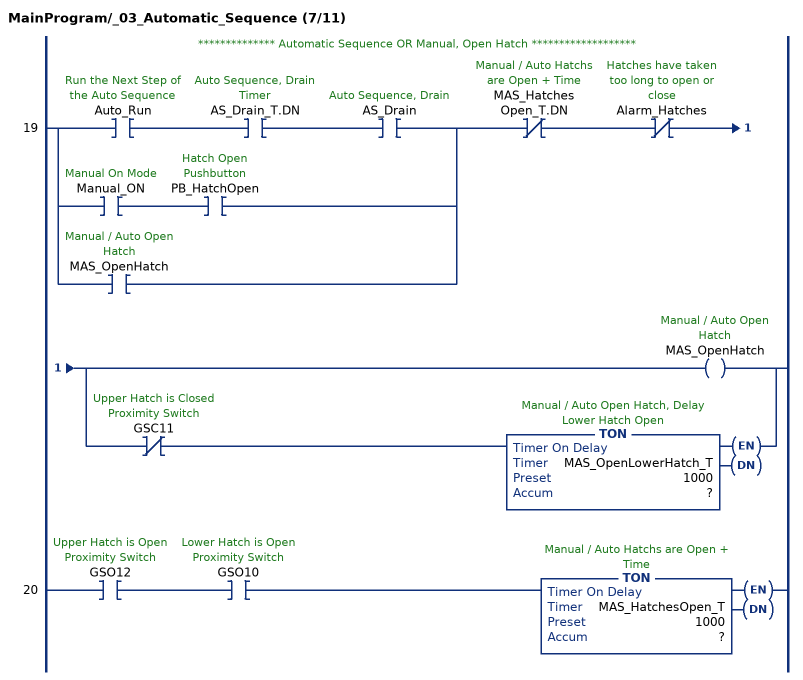
   // ************** Automatic Sequence OR Manual, Open Hatch *******************
   19: [XIC(Auto_Run) XIC(AS_Drain_T.DN) XIC(AS_Drain) ,XIC(Manual_ON) XIC(PB_HatchOpen) ,XIC(MAS_OpenHatch) ]XIO(MAS_HatchesOpen_T.DN)XIO(Alarm_Hatches)[OTE(MAS_OpenHatch) ,XIO(GSC11) TON(MAS_OpenLowerHatch_T,?,?) ];
   20: XIC(GSO12)XIC(GSO10)TON(MAS_HatchesOpen_T,?,?);
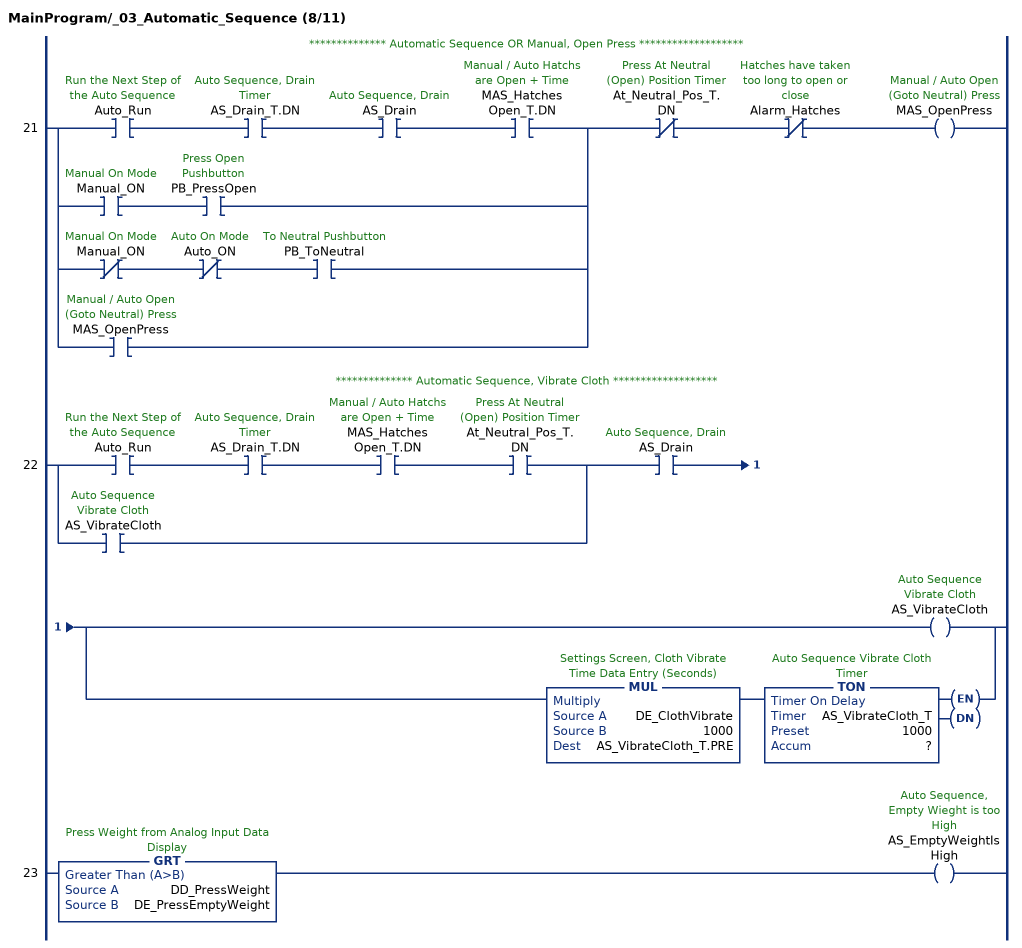
   // ************** Automatic Sequence OR Manual, Open Press *******************
   21: [XIC(Auto_Run) XIC(AS_Drain_T.DN) XIC(AS_Drain) XIC(MAS_HatchesOpen_T.DN) ,XIC(Manual_ON) XIC(PB_PressOpen) ,XIO(Manual_ON) XIO(Auto_ON) XIC(PB_ToNeutral) ,XIC(MAS_OpenPress) ]XIO(At_Neutral_Pos_T.DN)XIO(Alarm_Hatches)OTE(MAS_OpenPress);
   // ************** Automatic Sequence, Vibrate Cloth *******************
   22: [XIC(Auto_Run) XIC(AS_Drain_T.DN) XIC(MAS_HatchesOpen_T.DN) XIC(At_Neutral_Pos_T.DN) ,XIC(AS_VibrateCloth) ]XIC(AS_Drain)[OTE(AS_VibrateCloth) ,MUL(DE_ClothVibrate,1000,AS_VibrateCloth_T.PRE) TON(AS_VibrateCloth_T,?,?) ];
   23: GRT(DD_PressWeight,DE_PressEmptyWeight)OTE(AS_EmptyWeightIsHigh);
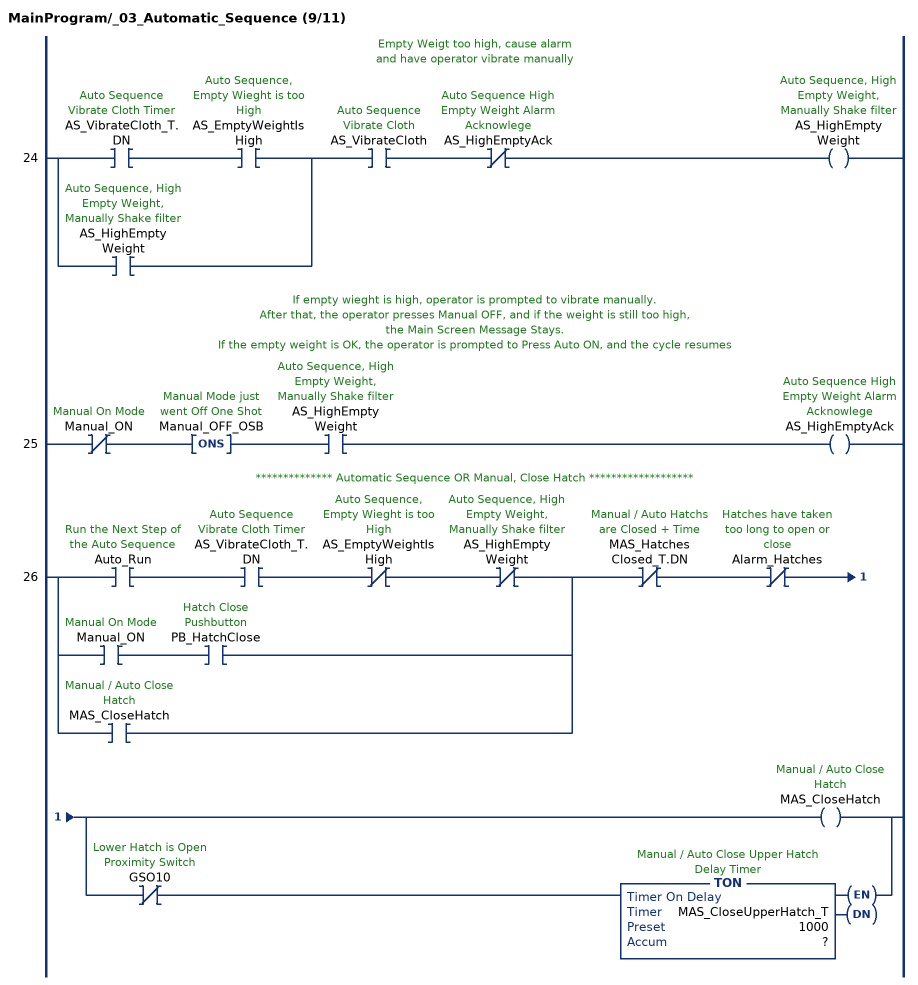
   // Empty Weigt too high, cause alarm
   // and have operator vibrate manually
   24: [XIC(AS_VibrateCloth_T.DN) XIC(AS_EmptyWeightIsHigh) ,XIC(AS_HighEmptyWeight) ]XIC(AS_VibrateCloth)XIO(AS_HighEmptyAck)OTE(AS_HighEmptyWeight);
   // If empty wieght is high, operator is prompted to vibrate manually.
   // After that, the operator presses Manual OFF, and if the weight is still too high,
   // the Main Screen Message Stays.
   // If the empty weight is OK, the operator is prompted to Press Auto ON, and the cycle resumes
   25: XIO(Manual_ON)ONS(Manual_OFF_OSB)XIC(AS_HighEmptyWeight)OTE(AS_HighEmptyAck);
   // ************** Automatic Sequence OR Manual, Close Hatch *******************
   26: [XIC(Auto_Run) XIC(AS_VibrateCloth_T.DN) XIO(AS_EmptyWeightIsHigh) XIO(AS_HighEmptyWeight) ,XIC(Manual_ON) XIC(PB_HatchClose) ,XIC(MAS_CloseHatch) ]XIO(MAS_HatchesClosed_T.DN)XIO(Alarm_Hatches)[OTE(MAS_CloseHatch) ,XIO(GSO10) TON(MAS_CloseUpperHatch_T,?,?) ];
